// TIA Portal V20 export
ORGANIZATION_BLOCK "Main"   // OB124, LAD, ProgramCycle
TITLE = "Main Program Sweep (Cycle)"
// stored: Namespace Conveyor2, SetENOAutomatically false
   VAR_INPUT
      Initial_Call : Bool;   // Initial call of this OB
      Remanence : Bool;   // =True, if remanent data are available
   END_VAR
BEGIN

REGION Network 1: Extra comment
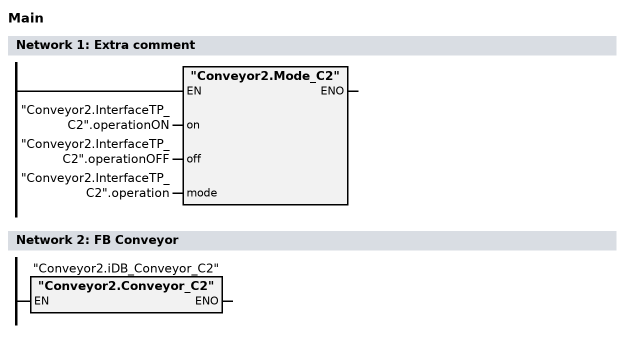
   RUNG wire#powerrail
      "Conveyor2.Mode_C2"(on := "Conveyor2.InterfaceTP_C2".operationON, off := "Conveyor2.InterfaceTP_C2".operationOFF, mode := "Conveyor2.InterfaceTP_C2".operation)
   END_RUNG
   // the same network as SCL:
   "Conveyor2.Mode_C2"(on := "Conveyor2.InterfaceTP_C2".operationON,
                       off := "Conveyor2.InterfaceTP_C2".operationOFF,
                       mode := "Conveyor2.InterfaceTP_C2".operation);
END_REGION

REGION Network 2: FB Conveyor
   RUNG wire#powerrail
      "Conveyor2.iDB_Conveyor_C2"()
   END_RUNG
   // the same network as SCL:
   "Conveyor2.iDB_Conveyor_C2"();   // "Conveyor2.Conveyor_C2"
END_REGION
END_ORGANIZATION_BLOCK
